{attribute 'qualified_only'}
{attribute 'strict'}
TYPE E_FunctionForkState :
(
	E_UNKNOWN,
	E_MOVING,
	E_CENTER, // HOME
	E_LEFT_COMPLETE,
	E_RIGHT_COMPLETE
);
END_TYPE

(* stored: Version 1.1.0.1, ProductVersion 3.1.4024.9
   DUT E_FunctionForkState: Id {2061d798-babc-46a1-9f31-39edf689236f} *)
